// TwinCAT 3 PLC project PLC
// ProgramVersion: 3.1.4026.19
// libraries:
//   Tc2_Standard, * (Beckhoff Automation GmbH)
//   Tc2_System, * (Beckhoff Automation GmbH)
//   Tc2_Utilities, * (Beckhoff Automation GmbH)
//   Tc3_EventLogger, * (Beckhoff Automation GmbH)
//   Tc3_Module, * (Beckhoff Automation GmbH)
// project tree:
//   / PlcTask.TcTTO
//   POUs/ MAIN.TcPOU
// real-time tasks:
//   TASK PlcTask: cycle T#10ms, priority 20, ADS port 350

CONFIGURATION PLC
    RESOURCE PLC ON TwinCAT3
        TASK PlcTask(INTERVAL := T#10ms, PRIORITY := 20);
        PROGRAM MAIN WITH PlcTask : MAIN;
    END_RESOURCE
END_CONFIGURATION

// ---- POUs/MAIN.TcPOU
PROGRAM MAIN
VAR
	TonDef:TON;
	wCount: WORD;
	
    bInit : BOOL := TRUE; 
    bSend : BOOL := TRUE; 

    fbMsg : FB_TcMessage; 
	fbTcEventLogger:FB_TcEventLogger;
	sLog:STRING;
	bExport:BOOL;
	fbTcEventCsvExportSettings: FB_TcEventCsvExportSettings;
	bExportError: BOOL;
	hrExportErrorCode: HRESULT;
	bExportResult: BOOL;
	sExportPath:STRING:='C:\TwinCAT\TEMP\';
	sFile:STRING:='Track.csv';
	sExportPathFile:STRING:='C:\TwinCAT\TEMP\Track.csv';
	fbNT_StartProcess: NT_StartProcess;
	sCommand:String;
	slog_IHM_Action:STRING:='Cold Start';
END_VAR

//Initialisation
IF bInit THEN
	wCount:=0;
    bInit := FALSE; 
    fbMsg.CreateEx(TC_EVENTS.EventClass.Logger, 0); 
END_IF

//On génénere un message log toute les 10s via l'alarme 'Log : ({0})'
TonDef(IN:= TRUE, PT:= T#10S, Q=> , ET=> );
IF TonDef.Q THEN
	wCount:=wCount+1;
	TonDef(IN:= FALSE);
	sLog:=concat('Event num: ',WORD_TO_STRING(wCount));	//Création du message
    fbMsg.ipArguments.Clear().AddString(sLog); //Enrichissement de l'argument {0}
	fbMsg.Send(0);//Envoie du message
END_IF


// On génére un evenement si sLog_IHM_Action est enrichi
IF slog_IHM_Action <>'' THEN
	fbMsg.ipArguments.Clear().AddString(slog_IHM_Action); //Enrichissement de l'argument {0}
	fbMsg.Send(0);//Envoie du message
	slog_IHM_Action:='';
END_IF



//Gestion de l'export
IF bExport THEN
	//Export au format CSV
	bExportResult:=fbTcEventLogger.ExportLoggedEvents(sFileName:=sExportPathFile , ipExportSettings:= fbTcEventCsvExportSettings, bError=> bExportError, hrErrorCode=>hrExportErrorCode );
	IF bExportResult THEN
		bExport:=FALSE;
	//Ouverture de l'explorateur
	sCommand:=CONCAT('C:\Windows\explorer.exe ',sExportPath);	
	fbNT_StartProcess(
		NETID:= '', 
		PATHSTR:= sCommand, 
		DIRNAME:= '', 
		COMNDLINE:= '', 
		START:= FALSE, //Front montant necessaire au bon fonctionnement
		TMOUT:= T#20S, 
		BUSY=> , 
		ERR=> , 
		ERRID=> );
	fbNT_StartProcess(START:= TRUE);
	END_IF
END_IF

END_PROGRAM
